Universal Robots PolyScope program: ur3_control.urp

Program test_socket_new (installation=default directory=/programs/usbdisk createdIn=5.9.4.1031232 lastSavedIn=3.14.3.1031232 robotSerialNumber=2017332543)
Calibrated DH parameters: a=[0.000031, -0.243823, -0.204309, 0.000009, -0.000019, 0]; d=[0.152052, 0.291789, 9.837334, -10.016486, 0.085275, 0.082255]; alpha=[1.569617, -0.005691, 0.006147, 1.57048, -1.570017, 0]; deltaTheta=[-0.000062, -0.006867, 0.302677, -0.295865, 0.000039, 0.000042]
BeforeStart
  Loop While (checkContinuously=false) expression=not socket_open("192.168.2.130",50002)
    Wait Sleep waitTime=0.05
  data := socket_read_ascii_float(6)
  If to_str(data[1])≟"nan"
    Script: socket_close()
    Halt
  desired_q := [data[1], data[2], data[3], data[4], data[5], data[6]]
  MoveJ speed 30 deg/s, acceleration 40 deg/s^2 (useActiveTCP=true)
    Waypoint Waypoint (Variable): variable=desired_q
  Wait Sleep waitTime=0.5
  current_p := get_actual_tcp_pose()
  desired_p := get_forward_kin(desired_q)
  If point_dist(current_p, desired_p) > 0.01
    Script: socket_send_string("Posicion no alcanzada")
    Script: socket_close()
    Halt
  Script: socket_send_string("Ready")
  Wait Sleep waitTime=0.05
Robot Program (runOnlyOnce=false)
  data := socket_read_ascii_float(6,timeout=5)
  If to_str(data[1])≟"nan"
    Script: socket_close()
    Halt
  desired_q := [data[1], data[2], data[3], data[4], data[5], data[6]]
  temp := get_actual_joint_positions()
  current_q := [temp[0], temp[1], temp[2], temp[3], temp[4], temp[5]]
  Script: socket_send_string(current_q)
Thread Thread_1 (runOnlyOnce=false)
  current_p := get_actual_tcp_pose()
  desired_p := get_forward_kin(desired_q)
  Script: servoj(desired_q,0,0,0.008,0.1,100)
